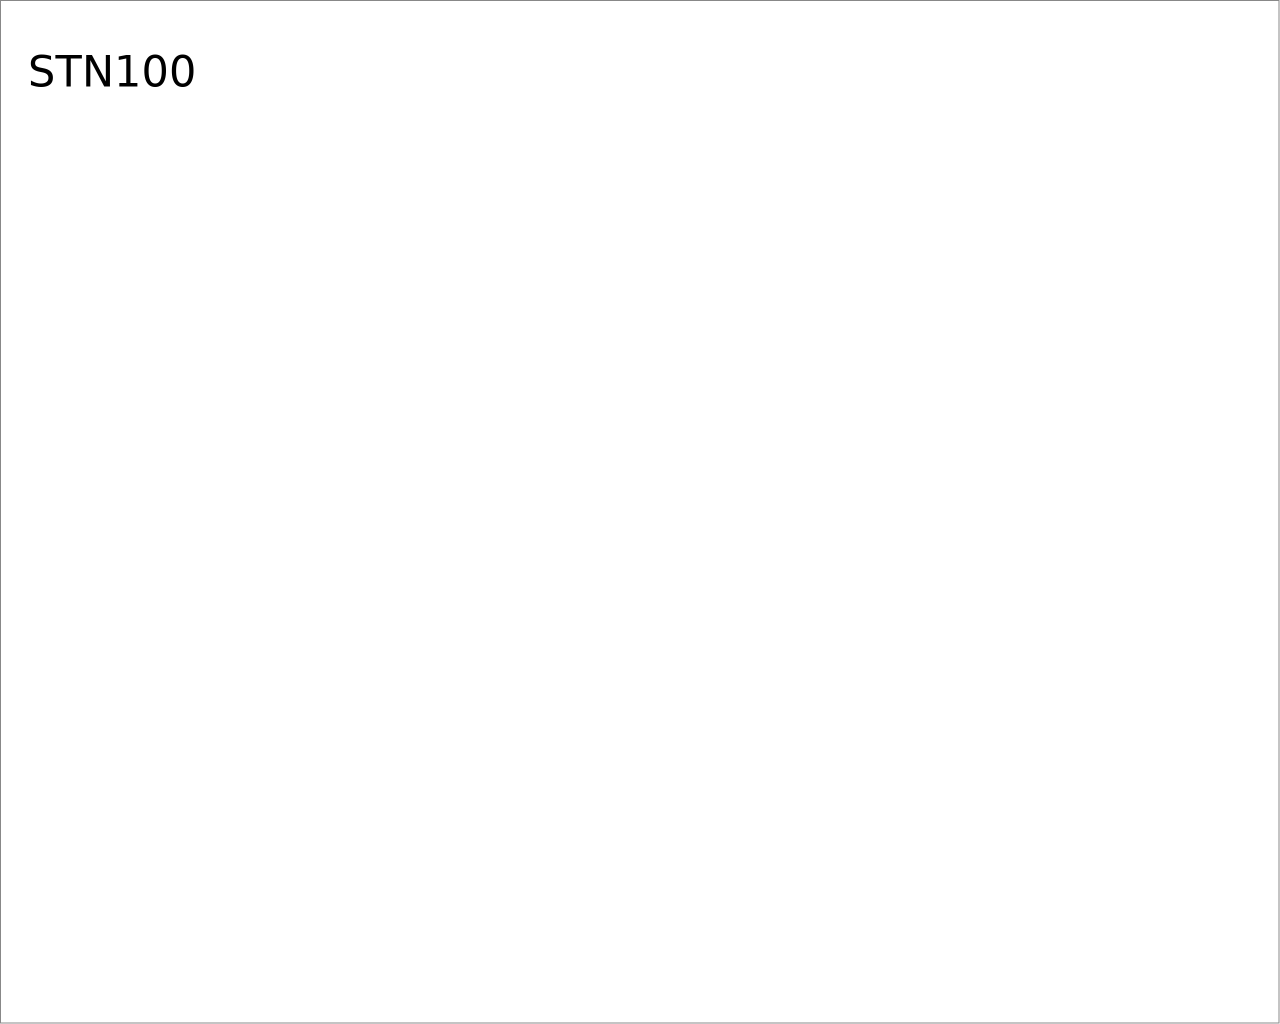
VISUALIZATION Visualization  // 1280x1024
    Label (16,29 193x85), "STN100"
END_VISUALIZATION

(* stored: Version 1.1.0.1, ProductVersion 3.1.4024.2
   Visu Visualization: Id {36610b8b-f765-4d79-bdc9-ce9f6f5c2cdd} *)
